FUNCTION_BLOCK FB_VariableSpeedMotor EXTENDS FB_VariableMotor

VAR
	fMotorSpeed : REAL;
END_VAR

METHOD M_SetSpeed : BOOL
VAR_INPUT
	fSpeedPercent : REAL;
END_VAR
fMotorSpeed := fSpeedPercent;
M_SetSpeed := TRUE;
END_METHOD

END_FUNCTION_BLOCK

(* stored: Version 1.1.0.1, ProductVersion 3.1.4024.16
   POU FB_VariableSpeedMotor: Id {630ec3ef-13ac-46cb-8e7d-096abd261b0e}, SpecialFunc None
   Method M_SetSpeed: Id {927d1fbb-148a-4705-87a1-0436e018022a} *)
